FUNCTION_BLOCK FB_Visu
VAR_INPUT
END_VAR
VAR_OUTPUT
END_VAR
VAR
END_VAR

visu.visuReceivedString:=MAIN.IV3.sStringFromReader;
visu.visuStingToBeSent:=MAIN.IV3.sStringToBeSend;
Visu.visuStatus:=MAIN.IV3.sStatus;

visu.visuError:=MAIN.IV3.bERROR;
Visu.visuStatusCommand:=main.IV3.sStatusCommand;
visu.visuStatusTCPIP:=main.IV3.sStatusTCPIP;
visu.visuStepCommand:=main.IV3.iStepCommands;
visu.visuStepTCPIP:=main.IV3.iStepTCPIP;
visu.visuTRigger:=main.btrigger;

END_FUNCTION_BLOCK

(* stored: Version 1.1.0.1, ProductVersion 3.1.4024.14
   POU FB_Visu: Id {1449b0d4-9f9a-4cc0-a1b8-c4105355c162}, SpecialFunc None *)
